SUBAPPLICATION Uebung_005 (* Subapplication Type *)
  (* Standard: 61499-2 *)
  (* Version 1.0, 2023-10-23, franz *)
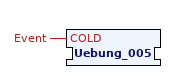
  EVENT_INPUT
    COLD;
  END_EVENT
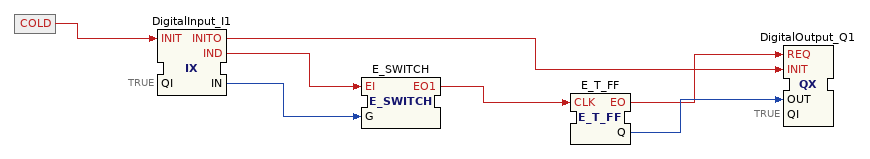
  FBS
    DigitalOutput_Q1 : QX(QI := TRUE);
    E_T_FF : E_T_FF;
    DigitalInput_I1 : IX(QI := TRUE);
    E_SWITCH : E_SWITCH;
  END_FBS
  EVENT_CONNECTIONS
    E_T_FF.EO TO DigitalOutput_Q1.REQ;
    COLD TO DigitalInput_I1.INIT;
    DigitalInput_I1.INITO TO DigitalOutput_Q1.INIT;
    DigitalInput_I1.IND TO E_SWITCH.EI;
    E_SWITCH.EO1 TO E_T_FF.CLK;
  END_CONNECTIONS
  DATA_CONNECTIONS
    E_T_FF.Q TO DigitalOutput_Q1.OUT;
    DigitalInput_I1.IN TO E_SWITCH.G;
  END_CONNECTIONS
END_SUBAPPLICATION
